(* Logix 5000 project; controller cal1632 1756-L62 rev 16.20; software revision 16.05; part 30 of 61 *)
(* tags used below, declared in another part *)
   AFI : BOOL;
   FAULT : BOOL;
   p01r02_plc_scan_time_in_sec : REAL;
   p01r09 : routine;
   p01r09_pb_global_reset : BOOL;
   p01r12_master_ramped_speed : REAL;
   p01r13_line_running : BOOL;
   p01r13_line_slow_ramp : BOOL;
   p01r13_permissive_drives : BOOL;
   p20_ai_lc01 : REAL;
   p20_ai_letoff_dia : REAL;
   p20_ai_lob_speed : REAL;
   p20_ao_lo_turret_selected_speed : REAL;
   p20_ao_lob_selected_speed : REAL;
   p20_ao_lob_torque : REAL;
   p20_di_clutch_prs_ok : BOOL;
   p20_di_lo_turret : acs800_di_normal;
   p20_di_lo_turret_therm : BOOL;
   p20_di_loa_active : BOOL;
   p20_di_lob_brake_thermostat : BOOL;
   p20_di_lob_fwd_dir : BOOL;
   p20_di_lob_jog : BOOL;
   p20_di_lob_motor_thermostat : BOOL;
   p20_di_lob_start : BOOL;
   p20_di_lob_stop : BOOL;
   p20_di_turret_fwd : BOOL;
   p20_di_turret_pos : BOOL;
   p20_di_turret_rev : BOOL;
   p20_do_close_nip : BOOL;
   p20_do_wdr_turret : acs800_do_normal;
   p20_param_high_accel_rate : REAL;
   p20_param_high_decel_rate : REAL;
   p20_param_jog_accel_rate : REAL;
   p20_param_jog_decel_rate : REAL;
   p20_param_letoff_jog_speed : REAL;
   p20_param_lo_turret_index_speed : REAL;
   p20_param_lof_fast_fill : REAL;
   p20_param_lof_slow_fill : REAL;
   p20_param_lof_stop_fill : REAL;
   p20_param_norm_accel_rate : REAL;
   p20_param_norm_decel_rate : REAL;
   p20_param_run_torque : REAL;
   p20_request_run_index_dir : BOOL;
   p20_request_run_index_rev_dir : BOOL;
   p20_vfd_di_lob : acs800_di_normal;
   p20_vfd_do_lob : acs800_do_normal;
   p20r10_speed_offset : REAL;
   p20r13_state : DINT;
   p20r15 : routine;
   p20r15_loa_on : BOOL;
   p20r15_request_tension : BOOL;
   p20r16 : routine;
   p20r16_loa_accel_decel_ramp : SYS_ACC_DEC_RAMP;
   p20r16_lob_accel : REAL;
   p20r16_lob_decel : REAL;
   p20r16_lob_on : BOOL;
   p20r16_lob_selected_speed : REAL;
   p20r16_permissive_run : BOOL;
   p20r16_request_jog_fwd : BOOL;
   p20r16_request_jog_rev : BOOL;
   p20r16_request_over_speed : BOOL;
   p20r16_request_position : BOOL;
   p20r16_request_stop : BOOL;
   p20r16_request_tension : BOOL;
   p20r16_request_thread_fwd : BOOL;
   p20r16_request_thread_rev : BOOL;
   p20r16_timer_fault : TIMER[10];
   p20r16_timer_warning : TIMER[4];
   p20r16_zero_speed : BOOL;
   p20r17 : routine;
   p20r17_ave_control : CONTROL;
   p20r17_diameter_clac_active : BOOL;
   p20r17_letoff_avg_diam_inch : REAL;
   p20r17_letoff_diam_avg_stack : REAL[20];
   p20r17_stack_ctrl : CONTROL;
   p20r17_timer : TIMER[5];
   p20r17_timer_fault : TIMER[5];
   p20r17_timer_warning : TIMER[5];
   p20r17_winder_a_unload : REAL;
   p20r18 : routine;
   p20r18_acc_dec_ramp : SYS_ACC_DEC_RAMP;
   p20r18_accel_rate : REAL;
   p20r18_decel_rate : REAL;
   p20r18_index_complete : BOOL;
   p20r18_index_move_timer : TIMER;
   p20r18_index_time : DINT;
   p20r18_index_time_offset : DINT;
   p20r18_index_timer : TIMER;
   p20r18_pb_index_fwd : BOOL;
   p20r18_pb_index_rev : BOOL;
   p20r18_permissive : BOOL;
   p20r18_request_index_fwd : BOOL;
   p20r18_request_index_rev : BOOL;
   p20r18_selected_speed : REAL;
   p20r18_timer_fault : TIMER[10];
   p20r18_timer_warning : TIMER[4];
   p20r18_zero_speed : BOOL;
   p22_ao_selected_speed : REAL;
   p22r11_request_thread_fwd : BOOL;
   p22r11_request_thread_rev : BOOL;
   p25r11_request_thread_fwd : BOOL;
   p25r11_request_thread_rev : BOOL;
(* P20_Letoff, continued *)

ROUTINE R16_Letoff_B_VFD   (* ladder *)
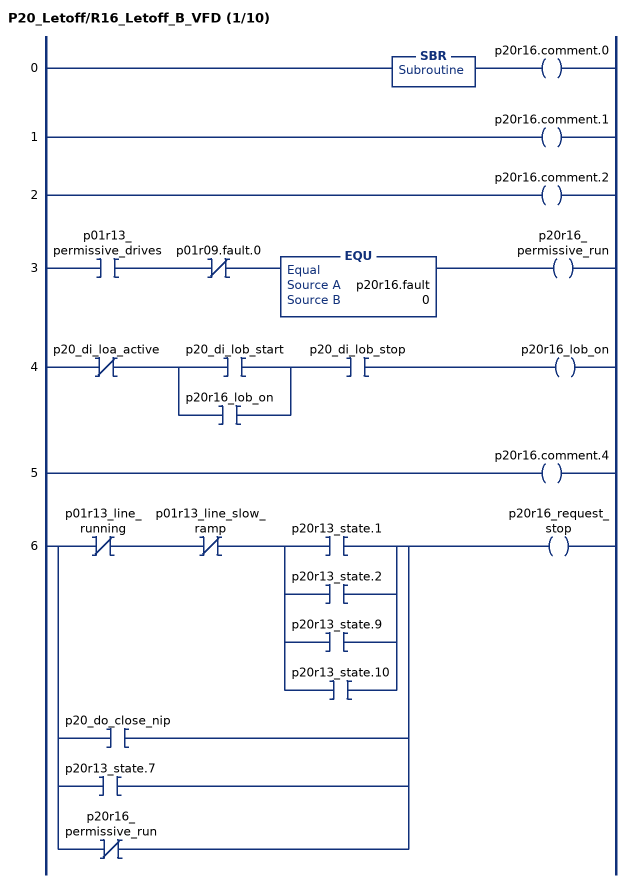
   0: SBR()OTE(p20r16.comment.0);
   1: OTE(p20r16.comment.1);
   2: OTE(p20r16.comment.2);
   3: XIC(p01r13_permissive_drives)XIO(p01r09.fault.0)EQU(p20r16.fault,0)OTE(p20r16_permissive_run);
   4: XIO(p20_di_loa_active)[XIC(p20_di_lob_start) ,XIC(p20r16_lob_on) ]XIC(p20_di_lob_stop)OTE(p20r16_lob_on);
   5: OTE(p20r16.comment.4);
   6: [XIO(p01r13_line_running) XIO(p01r13_line_slow_ramp) [XIC(p20r13_state.1) ,XIC(p20r13_state.2) ,XIC(p20r13_state.9) ,XIC(p20r13_state.10) ] ,XIC(p20_do_close_nip) ,XIC(p20r13_state.7) ,XIO(p20r16_permissive_run) ]OTE(p20r16_request_stop);
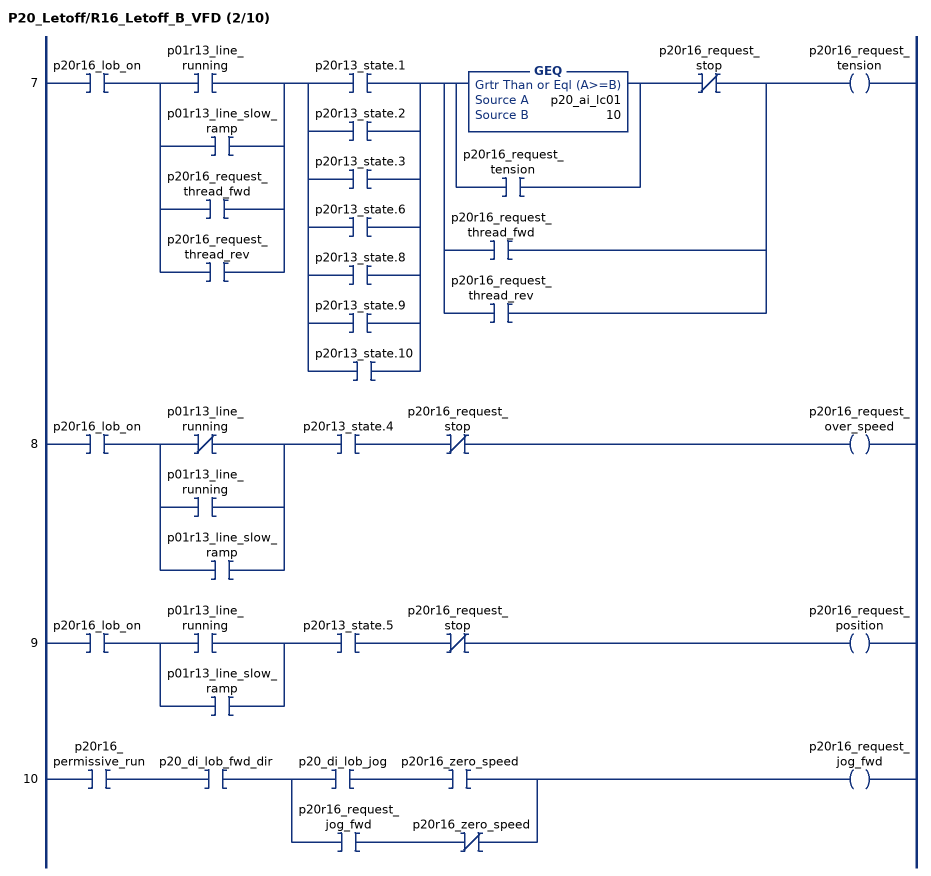
   7: XIC(p20r16_lob_on)[XIC(p01r13_line_running) ,XIC(p01r13_line_slow_ramp) ,XIC(p20r16_request_thread_fwd) ,XIC(p20r16_request_thread_rev) ][XIC(p20r13_state.1) ,XIC(p20r13_state.2) ,XIC(p20r13_state.3) ,XIC(p20r13_state.6) ,XIC(p20r13_state.8) ,XIC(p20r13_state.9) ,XIC(p20r13_state.10) ][[GEQ(p20_ai_lc01,10) ,XIC(p20r16_request_tension) ] XIO(p20r16_request_stop) ,XIC(p20r16_request_thread_fwd) ,XIC(p20r16_request_thread_rev) ]OTE(p20r16_request_tension);
   8: XIC(p20r16_lob_on)[XIO(p01r13_line_running) ,XIC(p01r13_line_running) ,XIC(p01r13_line_slow_ramp) ]XIC(p20r13_state.4)XIO(p20r16_request_stop)OTE(p20r16_request_over_speed);
   9: XIC(p20r16_lob_on)[XIC(p01r13_line_running) ,XIC(p01r13_line_slow_ramp) ]XIC(p20r13_state.5)XIO(p20r16_request_stop)OTE(p20r16_request_position);
   10: XIC(p20r16_permissive_run)XIC(p20_di_lob_fwd_dir)[XIC(p20_di_lob_jog) XIC(p20r16_zero_speed) ,XIC(p20r16_request_jog_fwd) XIO(p20r16_zero_speed) ]OTE(p20r16_request_jog_fwd);
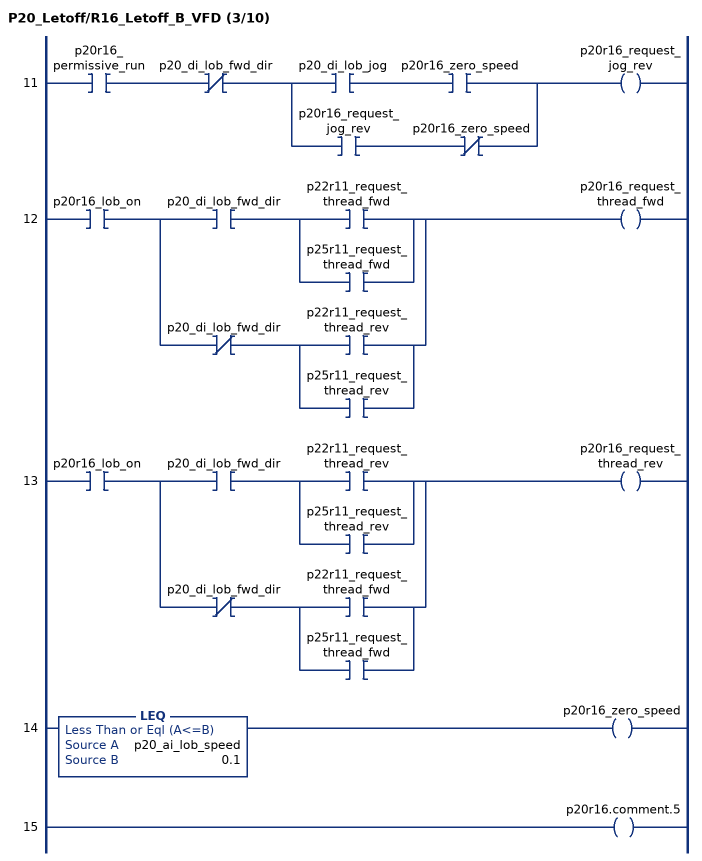
   11: XIC(p20r16_permissive_run)XIO(p20_di_lob_fwd_dir)[XIC(p20_di_lob_jog) XIC(p20r16_zero_speed) ,XIC(p20r16_request_jog_rev) XIO(p20r16_zero_speed) ]OTE(p20r16_request_jog_rev);
   12: XIC(p20r16_lob_on)[XIC(p20_di_lob_fwd_dir) [XIC(p22r11_request_thread_fwd) ,XIC(p25r11_request_thread_fwd) ] ,XIO(p20_di_lob_fwd_dir) [XIC(p22r11_request_thread_rev) ,XIC(p25r11_request_thread_rev) ] ]OTE(p20r16_request_thread_fwd);
   13: XIC(p20r16_lob_on)[XIC(p20_di_lob_fwd_dir) [XIC(p22r11_request_thread_rev) ,XIC(p25r11_request_thread_rev) ] ,XIO(p20_di_lob_fwd_dir) [XIC(p22r11_request_thread_fwd) ,XIC(p25r11_request_thread_fwd) ] ]OTE(p20r16_request_thread_rev);
   14: LEQ(p20_ai_lob_speed,0.1)OTE(p20r16_zero_speed);
   15: OTE(p20r16.comment.5);
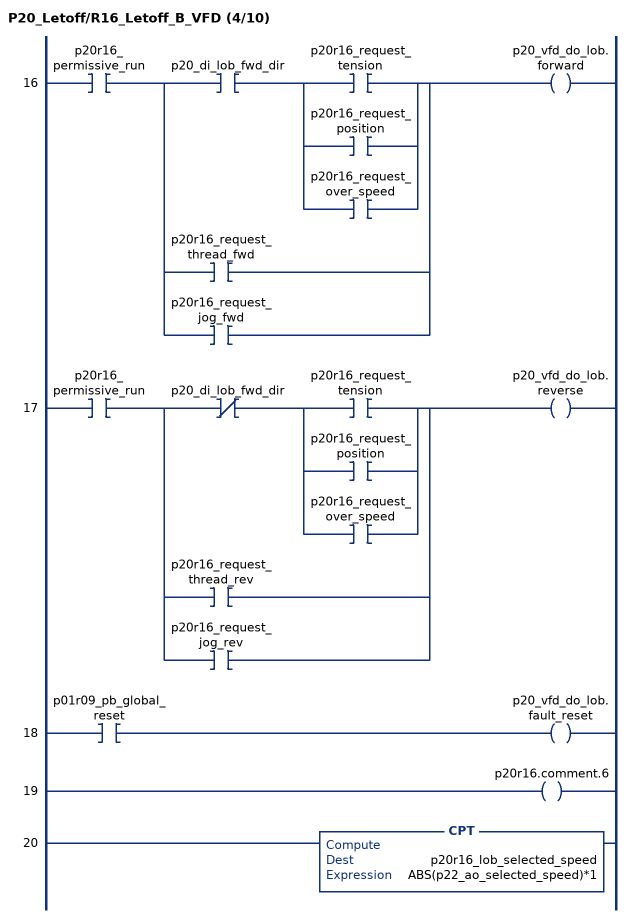
   16: XIC(p20r16_permissive_run)[XIC(p20_di_lob_fwd_dir) [XIC(p20r16_request_tension) ,XIC(p20r16_request_position) ,XIC(p20r16_request_over_speed) ] ,XIC(p20r16_request_thread_fwd) ,XIC(p20r16_request_jog_fwd) ]OTE(p20_vfd_do_lob.forward);
   17: XIC(p20r16_permissive_run)[XIO(p20_di_lob_fwd_dir) [XIC(p20r16_request_tension) ,XIC(p20r16_request_position) ,XIC(p20r16_request_over_speed) ] ,XIC(p20r16_request_thread_rev) ,XIC(p20r16_request_jog_rev) ]OTE(p20_vfd_do_lob.reverse);
   18: XIC(p01r09_pb_global_reset)OTE(p20_vfd_do_lob.fault_reset);
   19: OTE(p20r16.comment.6);
   20: CPT(p20r16_lob_selected_speed,ABS(p22_ao_selected_speed)*1);
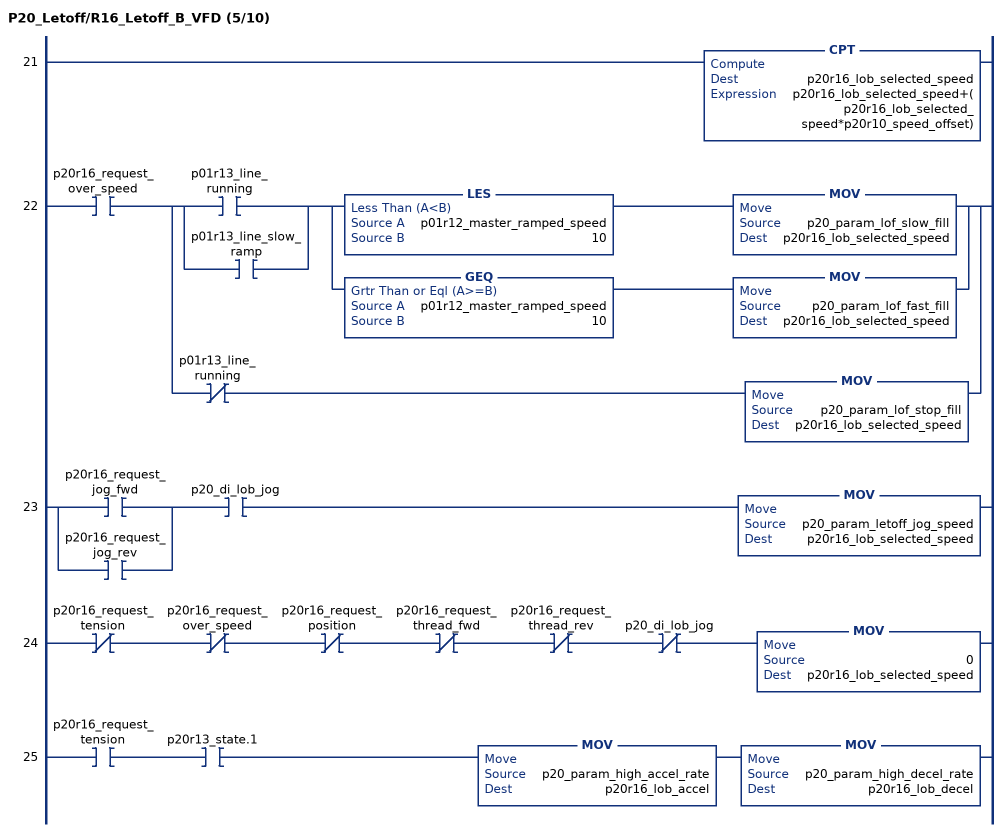
   21: CPT(p20r16_lob_selected_speed,p20r16_lob_selected_speed+(p20r16_lob_selected_speed*p20r10_speed_offset));
   22: XIC(p20r16_request_over_speed)[[XIC(p01r13_line_running) ,XIC(p01r13_line_slow_ramp) ] [LES(p01r12_master_ramped_speed,10) MOV(p20_param_lof_slow_fill,p20r16_lob_selected_speed) ,GEQ(p01r12_master_ramped_speed,10) MOV(p20_param_lof_fast_fill,p20r16_lob_selected_speed) ] ,XIO(p01r13_line_running) MOV(p20_param_lof_stop_fill,p20r16_lob_selected_speed) ];
   23: [XIC(p20r16_request_jog_fwd) ,XIC(p20r16_request_jog_rev) ]XIC(p20_di_lob_jog)MOV(p20_param_letoff_jog_speed,p20r16_lob_selected_speed);
   24: XIO(p20r16_request_tension)XIO(p20r16_request_over_speed)XIO(p20r16_request_position)XIO(p20r16_request_thread_fwd)XIO(p20r16_request_thread_rev)XIO(p20_di_lob_jog)MOV(0,p20r16_lob_selected_speed);
   25: XIC(p20r16_request_tension)XIC(p20r13_state.1)MOV(p20_param_high_accel_rate,p20r16_lob_accel)MOV(p20_param_high_decel_rate,p20r16_lob_decel);
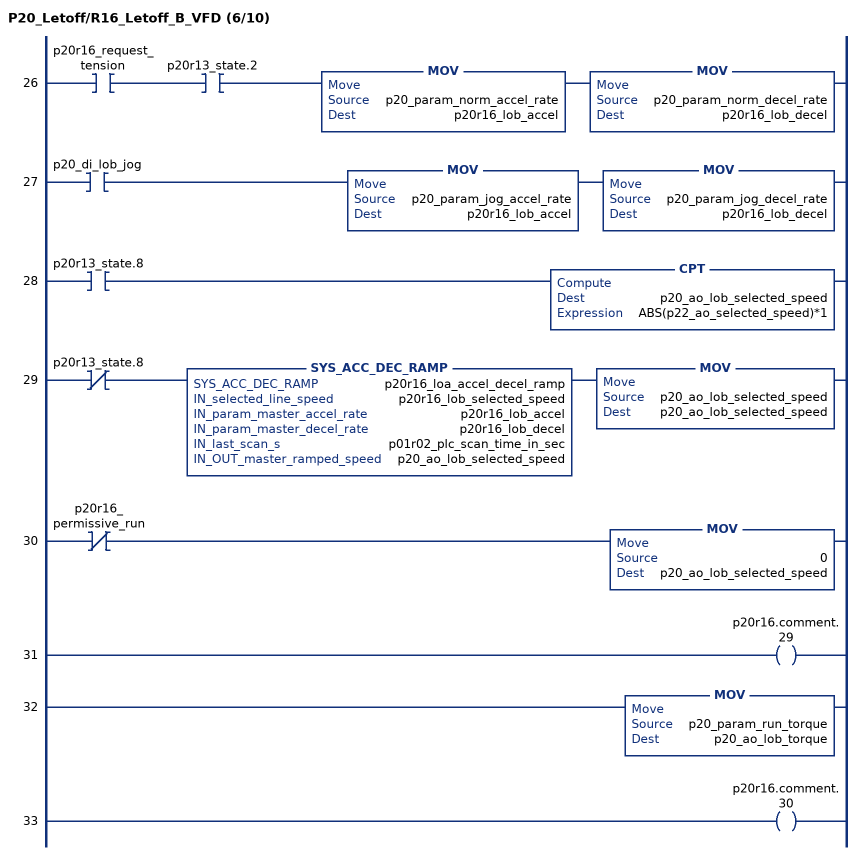
   26: XIC(p20r16_request_tension)XIC(p20r13_state.2)MOV(p20_param_norm_accel_rate,p20r16_lob_accel)MOV(p20_param_norm_decel_rate,p20r16_lob_decel);
   27: XIC(p20_di_lob_jog)MOV(p20_param_jog_accel_rate,p20r16_lob_accel)MOV(p20_param_jog_decel_rate,p20r16_lob_decel);
   28: XIC(p20r13_state.8)CPT(p20_ao_lob_selected_speed,ABS(p22_ao_selected_speed)*1);
   29: XIO(p20r13_state.8)SYS_ACC_DEC_RAMP(p20r16_loa_accel_decel_ramp,p20r16_lob_selected_speed,p20r16_lob_accel,p20r16_lob_decel,p01r02_plc_scan_time_in_sec,p20_ao_lob_selected_speed)MOV(p20_ao_lob_selected_speed,p20_ao_lob_selected_speed);
   30: XIO(p20r16_permissive_run)MOV(0,p20_ao_lob_selected_speed);
   31: OTE(p20r16.comment.29);
   32: MOV(p20_param_run_torque,p20_ao_lob_torque);
   33: OTE(p20r16.comment.30);
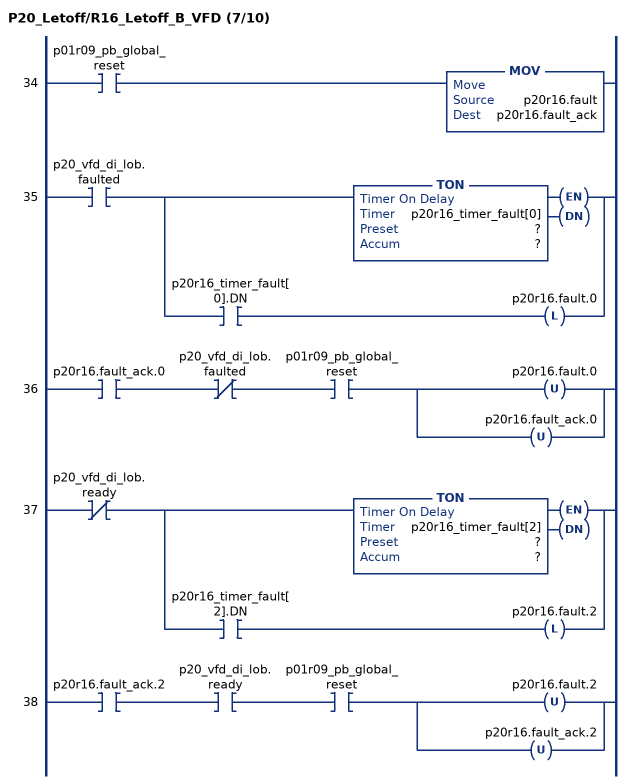
   34: XIC(p01r09_pb_global_reset)MOV(p20r16.fault,p20r16.fault_ack);
   35: XIC(p20_vfd_di_lob.faulted)[TON(p20r16_timer_fault[0],?,?) ,XIC(p20r16_timer_fault[0].DN) OTL(p20r16.fault.0) ];
   36: XIC(p20r16.fault_ack.0)XIO(p20_vfd_di_lob.faulted)XIC(p01r09_pb_global_reset)[OTU(p20r16.fault.0) ,OTU(p20r16.fault_ack.0) ];
   37: XIO(p20_vfd_di_lob.ready)[TON(p20r16_timer_fault[2],?,?) ,XIC(p20r16_timer_fault[2].DN) OTL(p20r16.fault.2) ];
   38: XIC(p20r16.fault_ack.2)XIC(p20_vfd_di_lob.ready)XIC(p01r09_pb_global_reset)[OTU(p20r16.fault.2) ,OTU(p20r16.fault_ack.2) ];
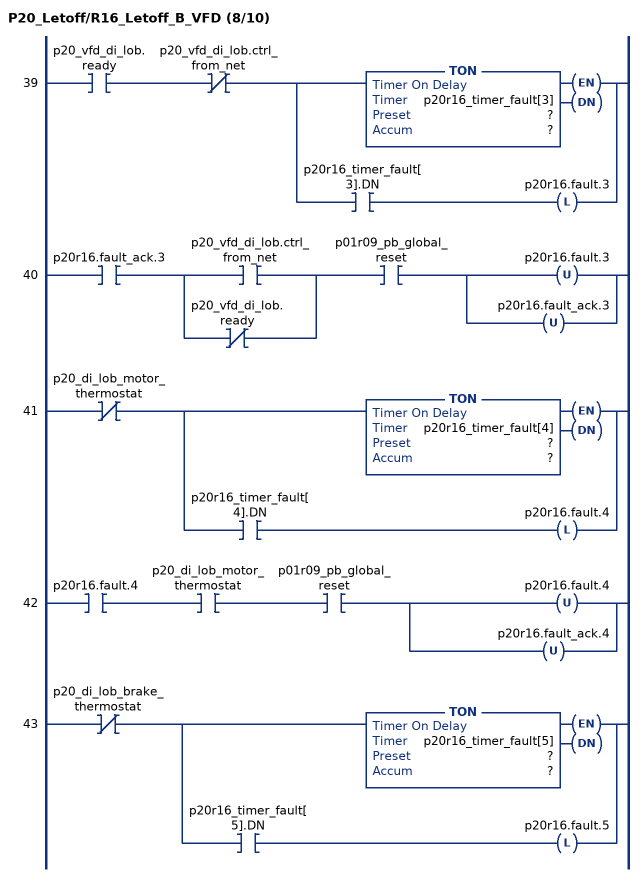
   39: XIC(p20_vfd_di_lob.ready)XIO(p20_vfd_di_lob.ctrl_from_net)[TON(p20r16_timer_fault[3],?,?) ,XIC(p20r16_timer_fault[3].DN) OTL(p20r16.fault.3) ];
   40: XIC(p20r16.fault_ack.3)[XIC(p20_vfd_di_lob.ctrl_from_net) ,XIO(p20_vfd_di_lob.ready) ]XIC(p01r09_pb_global_reset)[OTU(p20r16.fault.3) ,OTU(p20r16.fault_ack.3) ];
   41: XIO(p20_di_lob_motor_thermostat)[TON(p20r16_timer_fault[4],?,?) ,XIC(p20r16_timer_fault[4].DN) OTL(p20r16.fault.4) ];
   42: XIC(p20r16.fault.4)XIC(p20_di_lob_motor_thermostat)XIC(p01r09_pb_global_reset)[OTU(p20r16.fault.4) ,OTU(p20r16.fault_ack.4) ];
   43: XIO(p20_di_lob_brake_thermostat)[TON(p20r16_timer_fault[5],?,?) ,XIC(p20r16_timer_fault[5].DN) OTL(p20r16.fault.5) ];
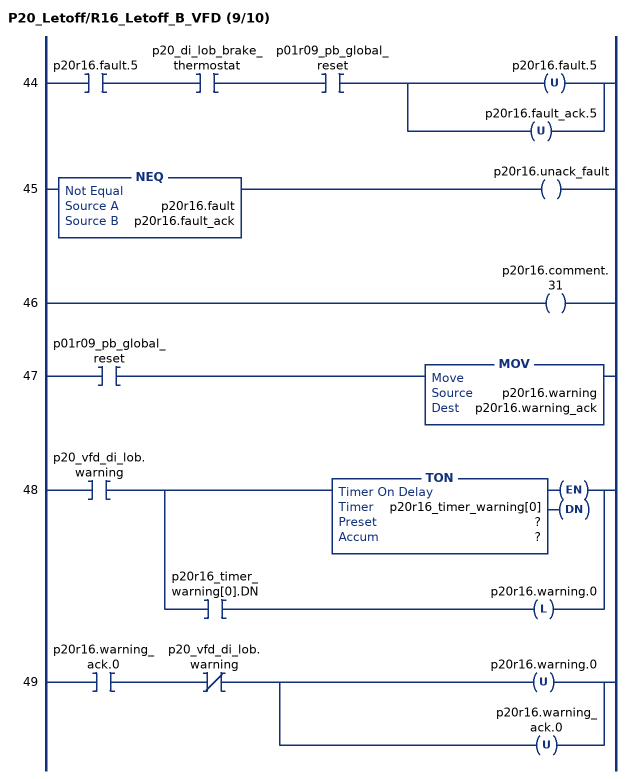
   44: XIC(p20r16.fault.5)XIC(p20_di_lob_brake_thermostat)XIC(p01r09_pb_global_reset)[OTU(p20r16.fault.5) ,OTU(p20r16.fault_ack.5) ];
   45: NEQ(p20r16.fault,p20r16.fault_ack)OTE(p20r16.unack_fault);
   46: OTE(p20r16.comment.31);
   47: XIC(p01r09_pb_global_reset)MOV(p20r16.warning,p20r16.warning_ack);
   48: XIC(p20_vfd_di_lob.warning)[TON(p20r16_timer_warning[0],?,?) ,XIC(p20r16_timer_warning[0].DN) OTL(p20r16.warning.0) ];
   49: XIC(p20r16.warning_ack.0)XIO(p20_vfd_di_lob.warning)[OTU(p20r16.warning.0) ,OTU(p20r16.warning_ack.0) ];
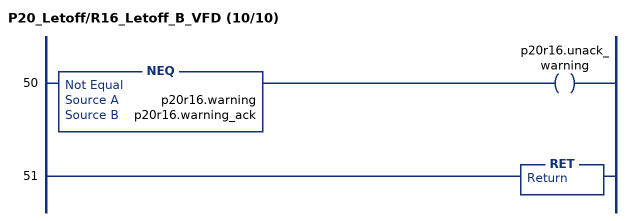
   50: NEQ(p20r16.warning,p20r16.warning_ack)OTE(p20r16.unack_warning);
   51: RET();
END_ROUTINE

ROUTINE R17_Letoff_Diameter_Calc   (* ladder *)
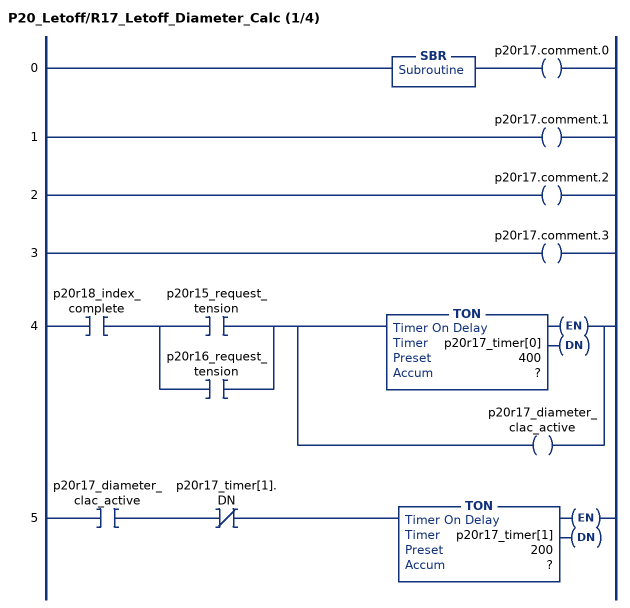
   0: SBR()OTE(p20r17.comment.0);
   1: OTE(p20r17.comment.1);
   2: OTE(p20r17.comment.2);
   3: OTE(p20r17.comment.3);
   4: XIC(p20r18_index_complete)[XIC(p20r15_request_tension) ,XIC(p20r16_request_tension) ][TON(p20r17_timer[0],?,?) ,OTE(p20r17_diameter_clac_active) ];
   5: XIC(p20r17_diameter_clac_active)XIO(p20r17_timer[1].DN)TON(p20r17_timer[1],?,?);
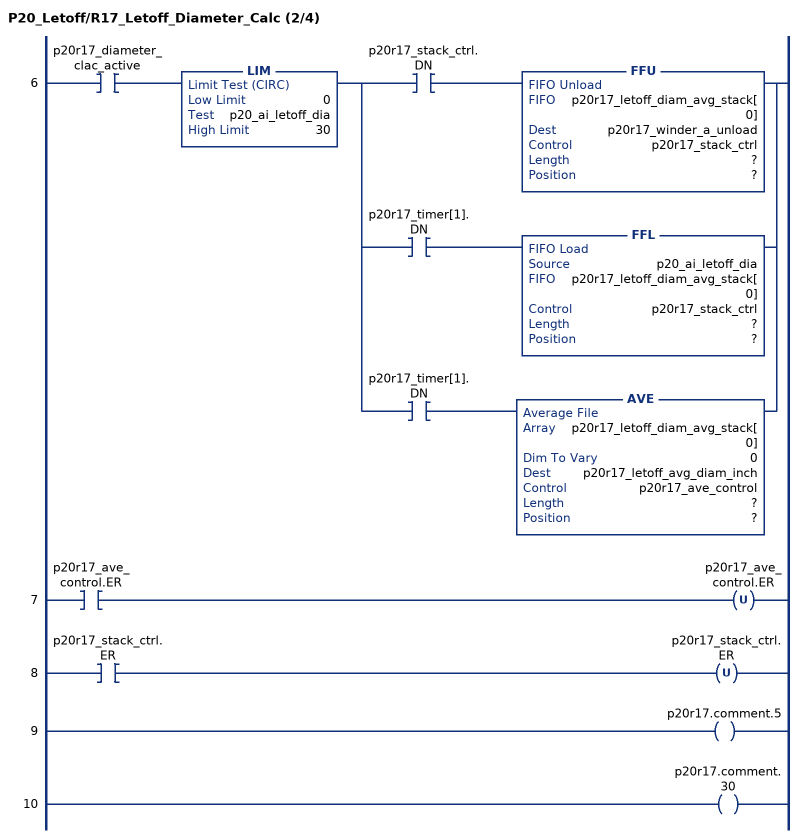
   6: XIC(p20r17_diameter_clac_active)LIM(0,p20_ai_letoff_dia,30)[XIC(p20r17_stack_ctrl.DN) FFU(p20r17_letoff_diam_avg_stack[0],p20r17_winder_a_unload,p20r17_stack_ctrl,?,?) ,XIC(p20r17_timer[1].DN) FFL(p20_ai_letoff_dia,p20r17_letoff_diam_avg_stack[0],p20r17_stack_ctrl,?,?) ,XIC(p20r17_timer[1].DN) AVE(p20r17_letoff_diam_avg_stack[0],0,p20r17_letoff_avg_diam_inch,p20r17_ave_control,?,?) ];
   7: XIC(p20r17_ave_control.ER)OTU(p20r17_ave_control.ER);
   8: XIC(p20r17_stack_ctrl.ER)OTU(p20r17_stack_ctrl.ER);
   9: OTE(p20r17.comment.5);
   10: OTE(p20r17.comment.30);
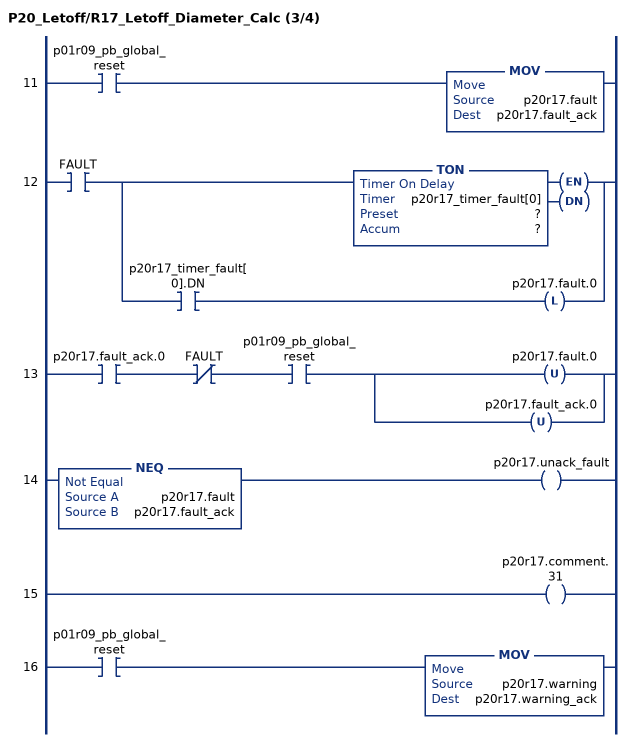
   11: XIC(p01r09_pb_global_reset)MOV(p20r17.fault,p20r17.fault_ack);
   12: XIC(FAULT)[TON(p20r17_timer_fault[0],?,?) ,XIC(p20r17_timer_fault[0].DN) OTL(p20r17.fault.0) ];
   13: XIC(p20r17.fault_ack.0)XIO(FAULT)XIC(p01r09_pb_global_reset)[OTU(p20r17.fault.0) ,OTU(p20r17.fault_ack.0) ];
   14: NEQ(p20r17.fault,p20r17.fault_ack)OTE(p20r17.unack_fault);
   15: OTE(p20r17.comment.31);
   16: XIC(p01r09_pb_global_reset)MOV(p20r17.warning,p20r17.warning_ack);
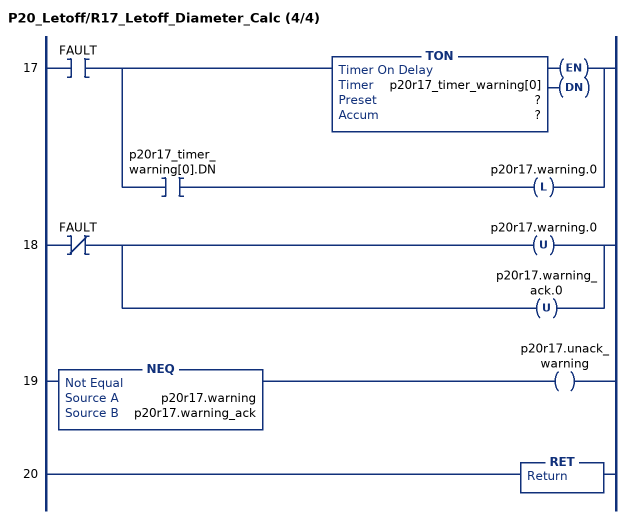
   17: XIC(FAULT)[TON(p20r17_timer_warning[0],?,?) ,XIC(p20r17_timer_warning[0].DN) OTL(p20r17.warning.0) ];
   18: XIO(FAULT)[OTU(p20r17.warning.0) ,OTU(p20r17.warning_ack.0) ];
   19: NEQ(p20r17.warning,p20r17.warning_ack)OTE(p20r17.unack_warning);
   20: RET();
END_ROUTINE

ROUTINE R18_Letoff_Turret_VFD   (* ladder *)
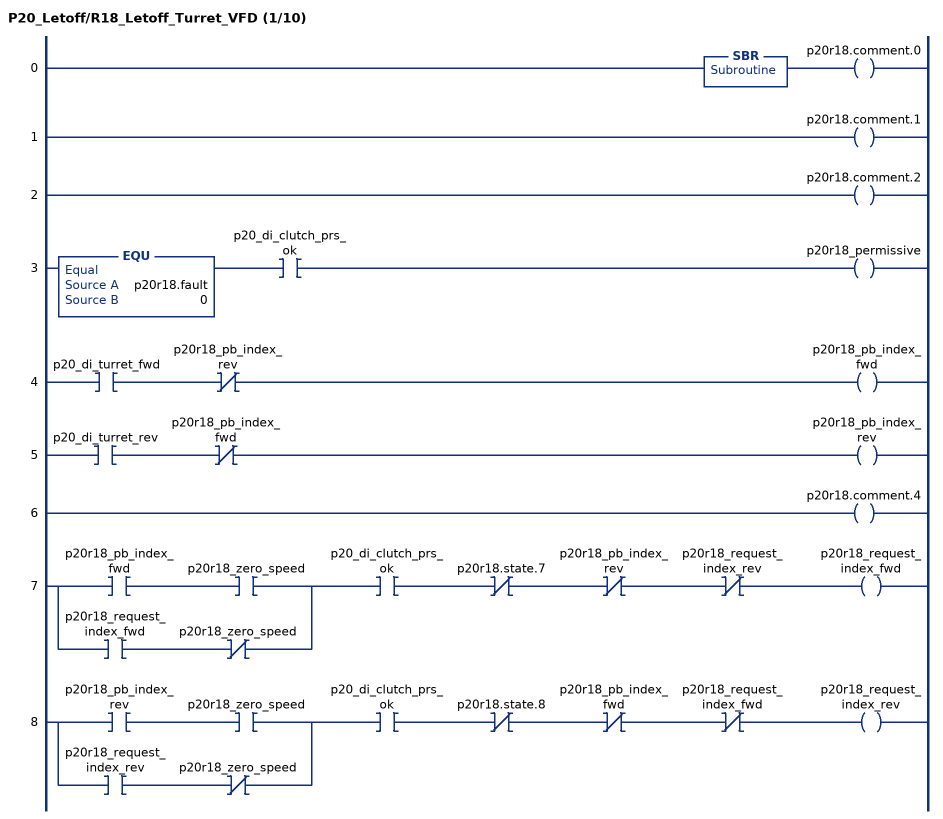
   0: SBR()OTE(p20r18.comment.0);
   1: OTE(p20r18.comment.1);
   2: OTE(p20r18.comment.2);
   3: EQU(p20r18.fault,0)XIC(p20_di_clutch_prs_ok)OTE(p20r18_permissive);
   4: XIC(p20_di_turret_fwd)XIO(p20r18_pb_index_rev)OTE(p20r18_pb_index_fwd);
   5: XIC(p20_di_turret_rev)XIO(p20r18_pb_index_fwd)OTE(p20r18_pb_index_rev);
   6: OTE(p20r18.comment.4);
   7: [XIC(p20r18_pb_index_fwd) XIC(p20r18_zero_speed) ,XIC(p20r18_request_index_fwd) XIO(p20r18_zero_speed) ]XIC(p20_di_clutch_prs_ok)XIO(p20r18.state.7)XIO(p20r18_pb_index_rev)XIO(p20r18_request_index_rev)OTE(p20r18_request_index_fwd);
   8: [XIC(p20r18_pb_index_rev) XIC(p20r18_zero_speed) ,XIC(p20r18_request_index_rev) XIO(p20r18_zero_speed) ]XIC(p20_di_clutch_prs_ok)XIO(p20r18.state.8)XIO(p20r18_pb_index_fwd)XIO(p20r18_request_index_fwd)OTE(p20r18_request_index_rev);
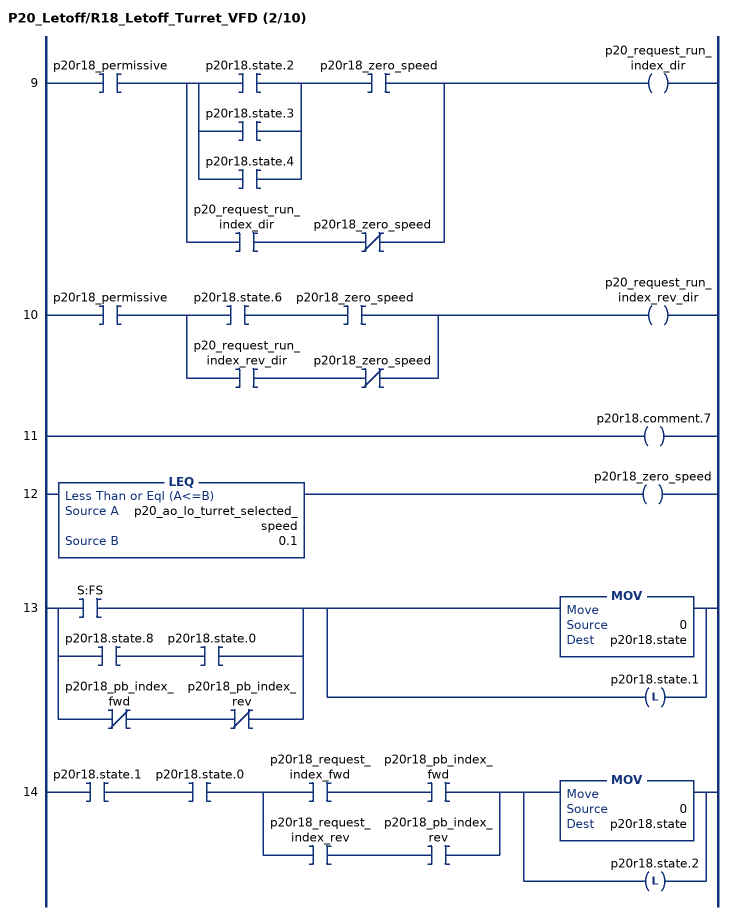
   9: XIC(p20r18_permissive)[[XIC(p20r18.state.2) ,XIC(p20r18.state.3) ,XIC(p20r18.state.4) ] XIC(p20r18_zero_speed) ,XIC(p20_request_run_index_dir) XIO(p20r18_zero_speed) ]OTE(p20_request_run_index_dir);
   10: XIC(p20r18_permissive)[XIC(p20r18.state.6) XIC(p20r18_zero_speed) ,XIC(p20_request_run_index_rev_dir) XIO(p20r18_zero_speed) ]OTE(p20_request_run_index_rev_dir);
   11: OTE(p20r18.comment.7);
   12: LEQ(p20_ao_lo_turret_selected_speed,0.1)OTE(p20r18_zero_speed);
   13: [XIC(S:FS) ,XIC(p20r18.state.8) XIC(p20r18.state.0) ,XIO(p20r18_pb_index_fwd) XIO(p20r18_pb_index_rev) ][MOV(0,p20r18.state) ,OTL(p20r18.state.1) ];
   14: XIC(p20r18.state.1)XIC(p20r18.state.0)[XIC(p20r18_request_index_fwd) XIC(p20r18_pb_index_fwd) ,XIC(p20r18_request_index_rev) XIC(p20r18_pb_index_rev) ][MOV(0,p20r18.state) ,OTL(p20r18.state.2) ];
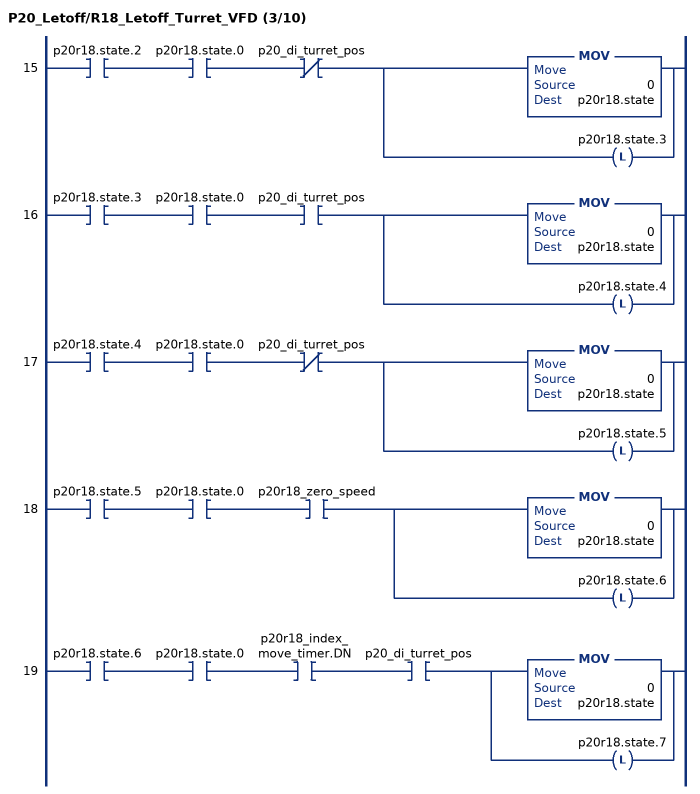
   15: XIC(p20r18.state.2)XIC(p20r18.state.0)XIO(p20_di_turret_pos)[MOV(0,p20r18.state) ,OTL(p20r18.state.3) ];
   16: XIC(p20r18.state.3)XIC(p20r18.state.0)XIC(p20_di_turret_pos)[MOV(0,p20r18.state) ,OTL(p20r18.state.4) ];
   17: XIC(p20r18.state.4)XIC(p20r18.state.0)XIO(p20_di_turret_pos)[MOV(0,p20r18.state) ,OTL(p20r18.state.5) ];
   18: XIC(p20r18.state.5)XIC(p20r18.state.0)XIC(p20r18_zero_speed)[MOV(0,p20r18.state) ,OTL(p20r18.state.6) ];
   19: XIC(p20r18.state.6)XIC(p20r18.state.0)XIC(p20r18_index_move_timer.DN)XIC(p20_di_turret_pos)[MOV(0,p20r18.state) ,OTL(p20r18.state.7) ];
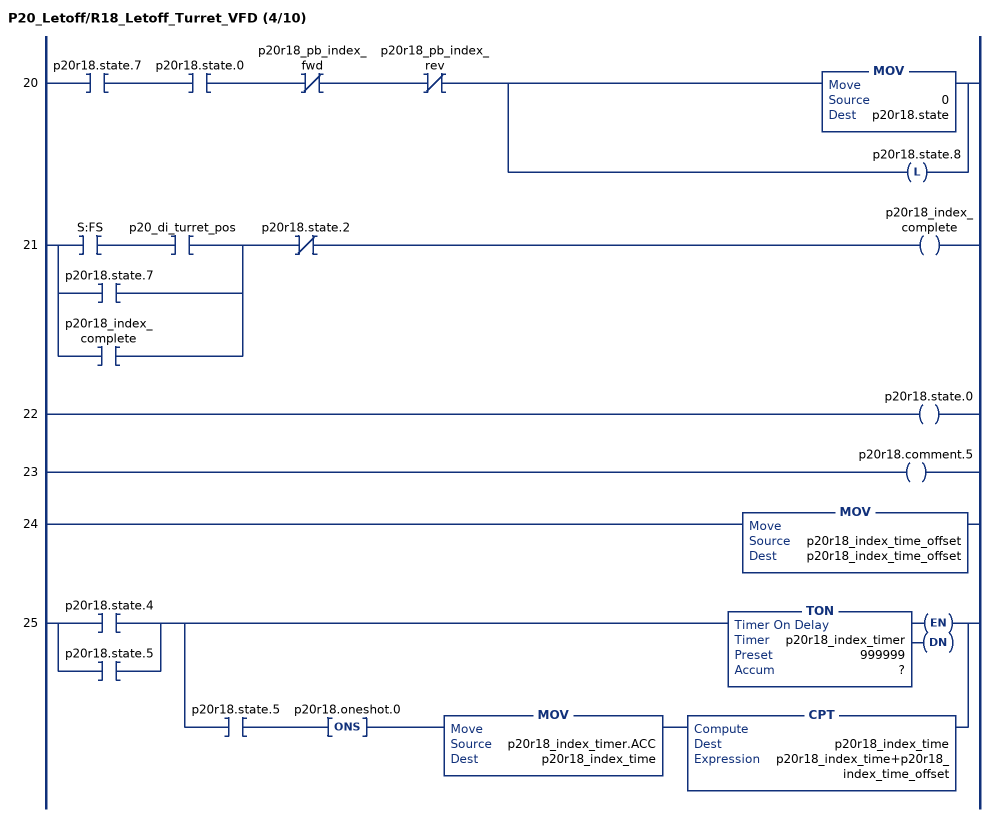
   20: XIC(p20r18.state.7)XIC(p20r18.state.0)XIO(p20r18_pb_index_fwd)XIO(p20r18_pb_index_rev)[MOV(0,p20r18.state) ,OTL(p20r18.state.8) ];
   21: [XIC(S:FS) XIC(p20_di_turret_pos) ,XIC(p20r18.state.7) ,XIC(p20r18_index_complete) ]XIO(p20r18.state.2)OTE(p20r18_index_complete);
   22: OTE(p20r18.state.0);
   23: OTE(p20r18.comment.5);
   24: MOV(p20r18_index_time_offset,p20r18_index_time_offset);
   25: [XIC(p20r18.state.4) ,XIC(p20r18.state.5) ][TON(p20r18_index_timer,?,?) ,XIC(p20r18.state.5) ONS(p20r18.oneshot.0) MOV(p20r18_index_timer.ACC,p20r18_index_time) CPT(p20r18_index_time,p20r18_index_time+p20r18_index_time_offset) ];
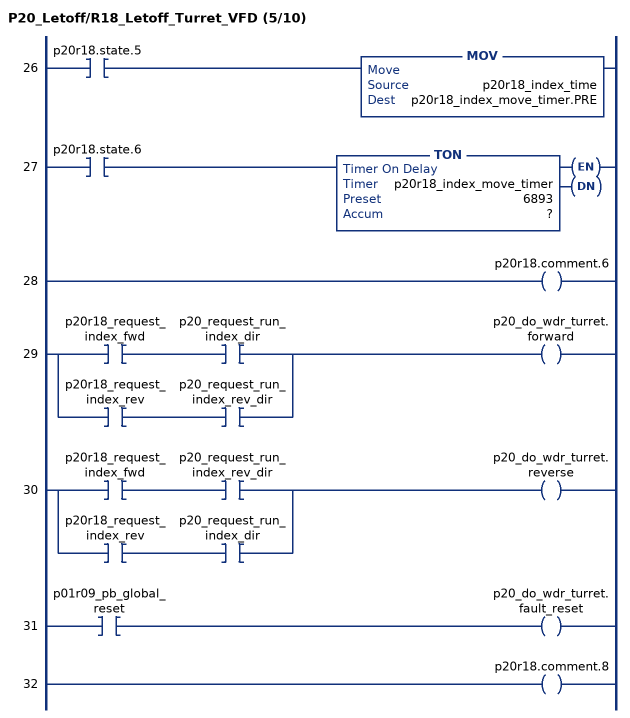
   26: XIC(p20r18.state.5)MOV(p20r18_index_time,p20r18_index_move_timer.PRE);
   27: XIC(p20r18.state.6)TON(p20r18_index_move_timer,?,?);
   28: OTE(p20r18.comment.6);
   29: [XIC(p20r18_request_index_fwd) XIC(p20_request_run_index_dir) ,XIC(p20r18_request_index_rev) XIC(p20_request_run_index_rev_dir) ]OTE(p20_do_wdr_turret.forward);
   30: [XIC(p20r18_request_index_fwd) XIC(p20_request_run_index_rev_dir) ,XIC(p20r18_request_index_rev) XIC(p20_request_run_index_dir) ]OTE(p20_do_wdr_turret.reverse);
   31: XIC(p01r09_pb_global_reset)OTE(p20_do_wdr_turret.fault_reset);
   32: OTE(p20r18.comment.8);
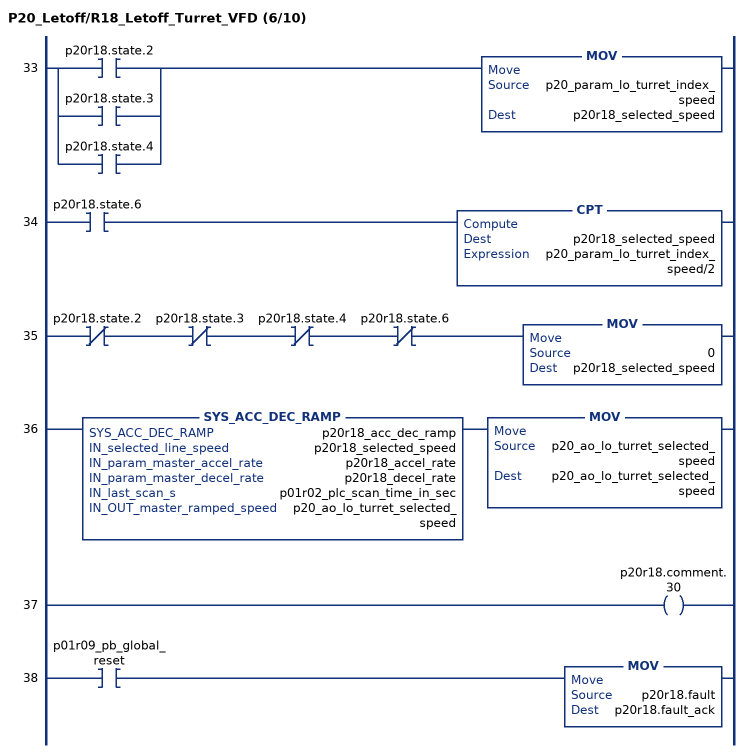
   33: [XIC(p20r18.state.2) ,XIC(p20r18.state.3) ,XIC(p20r18.state.4) ]MOV(p20_param_lo_turret_index_speed,p20r18_selected_speed);
   34: XIC(p20r18.state.6)CPT(p20r18_selected_speed,p20_param_lo_turret_index_speed/2);
   35: XIO(p20r18.state.2)XIO(p20r18.state.3)XIO(p20r18.state.4)XIO(p20r18.state.6)MOV(0,p20r18_selected_speed);
   36: SYS_ACC_DEC_RAMP(p20r18_acc_dec_ramp,p20r18_selected_speed,p20r18_accel_rate,p20r18_decel_rate,p01r02_plc_scan_time_in_sec,p20_ao_lo_turret_selected_speed)MOV(p20_ao_lo_turret_selected_speed,p20_ao_lo_turret_selected_speed);
   37: OTE(p20r18.comment.30);
   38: XIC(p01r09_pb_global_reset)MOV(p20r18.fault,p20r18.fault_ack);
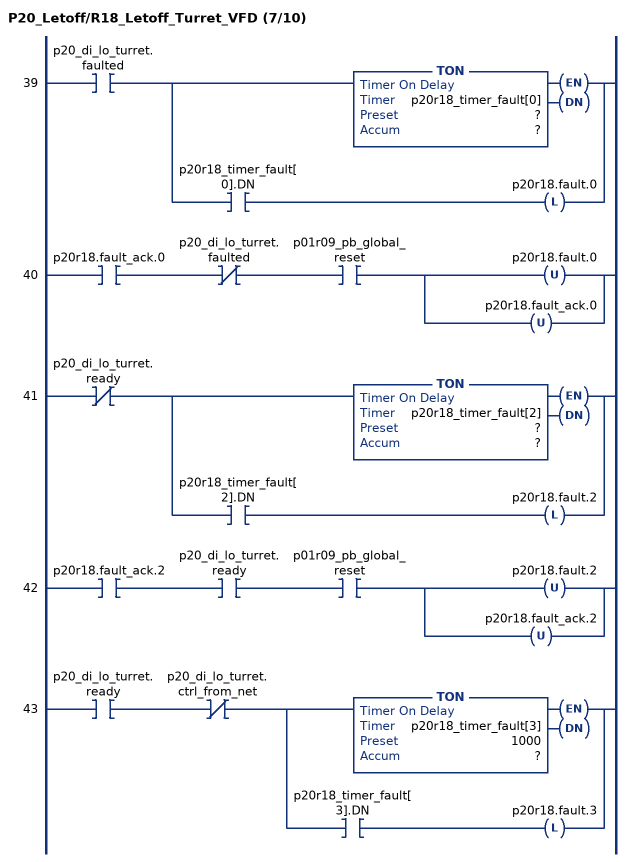
   39: XIC(p20_di_lo_turret.faulted)[TON(p20r18_timer_fault[0],?,?) ,XIC(p20r18_timer_fault[0].DN) OTL(p20r18.fault.0) ];
   40: XIC(p20r18.fault_ack.0)XIO(p20_di_lo_turret.faulted)XIC(p01r09_pb_global_reset)[OTU(p20r18.fault.0) ,OTU(p20r18.fault_ack.0) ];
   41: XIO(p20_di_lo_turret.ready)[TON(p20r18_timer_fault[2],?,?) ,XIC(p20r18_timer_fault[2].DN) OTL(p20r18.fault.2) ];
   42: XIC(p20r18.fault_ack.2)XIC(p20_di_lo_turret.ready)XIC(p01r09_pb_global_reset)[OTU(p20r18.fault.2) ,OTU(p20r18.fault_ack.2) ];
   43: XIC(p20_di_lo_turret.ready)XIO(p20_di_lo_turret.ctrl_from_net)[TON(p20r18_timer_fault[3],?,?) ,XIC(p20r18_timer_fault[3].DN) OTL(p20r18.fault.3) ];
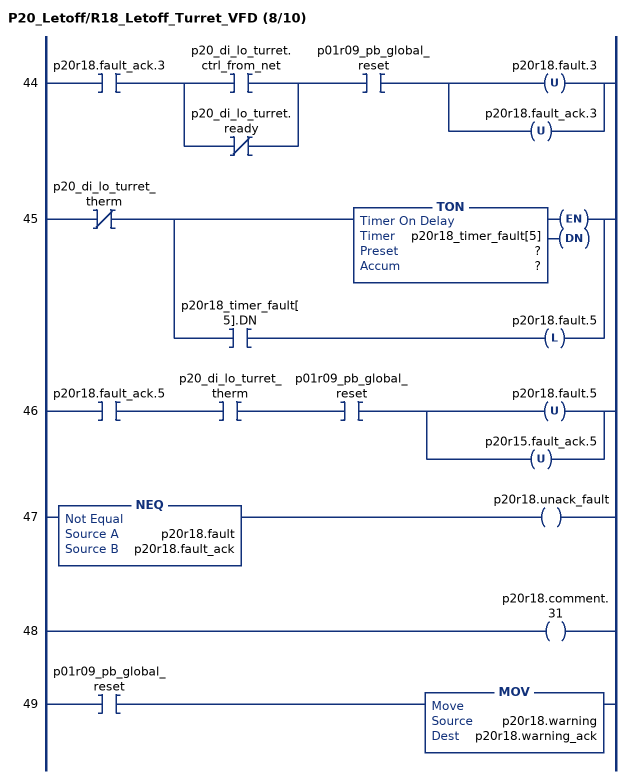
   44: XIC(p20r18.fault_ack.3)[XIC(p20_di_lo_turret.ctrl_from_net) ,XIO(p20_di_lo_turret.ready) ]XIC(p01r09_pb_global_reset)[OTU(p20r18.fault.3) ,OTU(p20r18.fault_ack.3) ];
   45: XIO(p20_di_lo_turret_therm)[TON(p20r18_timer_fault[5],?,?) ,XIC(p20r18_timer_fault[5].DN) OTL(p20r18.fault.5) ];
   46: XIC(p20r18.fault_ack.5)XIC(p20_di_lo_turret_therm)XIC(p01r09_pb_global_reset)[OTU(p20r18.fault.5) ,OTU(p20r15.fault_ack.5) ];
   47: NEQ(p20r18.fault,p20r18.fault_ack)OTE(p20r18.unack_fault);
   48: OTE(p20r18.comment.31);
   49: XIC(p01r09_pb_global_reset)MOV(p20r18.warning,p20r18.warning_ack);
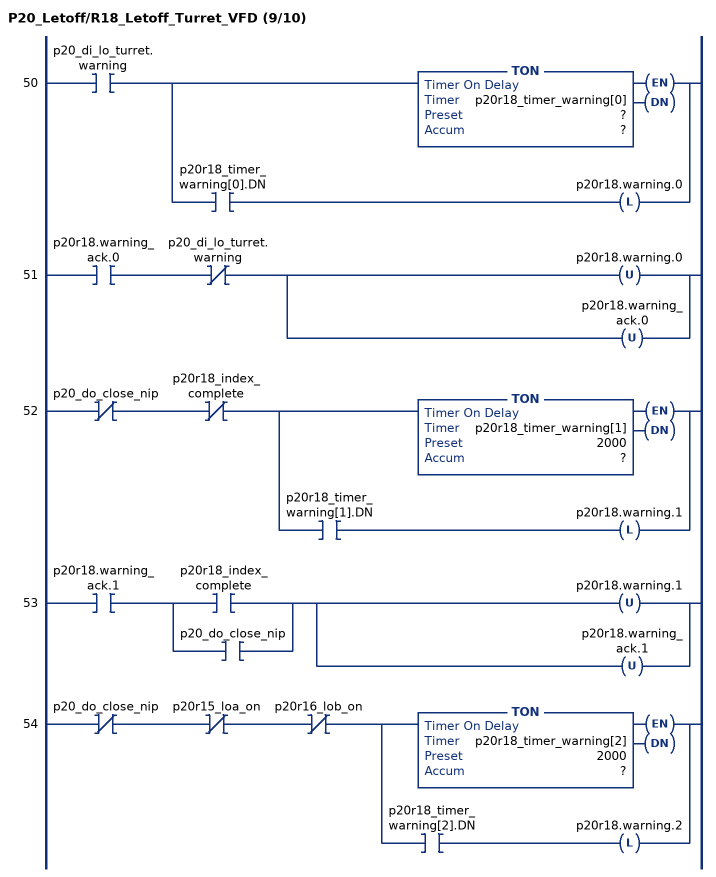
   50: XIC(p20_di_lo_turret.warning)[TON(p20r18_timer_warning[0],?,?) ,XIC(p20r18_timer_warning[0].DN) OTL(p20r18.warning.0) ];
   51: XIC(p20r18.warning_ack.0)XIO(p20_di_lo_turret.warning)[OTU(p20r18.warning.0) ,OTU(p20r18.warning_ack.0) ];
   52: XIO(p20_do_close_nip)XIO(p20r18_index_complete)[TON(p20r18_timer_warning[1],?,?) ,XIC(p20r18_timer_warning[1].DN) OTL(p20r18.warning.1) ];
   53: XIC(p20r18.warning_ack.1)[XIC(p20r18_index_complete) ,XIC(p20_do_close_nip) ][OTU(p20r18.warning.1) ,OTU(p20r18.warning_ack.1) ];
   54: XIO(p20_do_close_nip)XIO(p20r15_loa_on)XIO(p20r16_lob_on)[TON(p20r18_timer_warning[2],?,?) ,XIC(p20r18_timer_warning[2].DN) OTL(p20r18.warning.2) ];
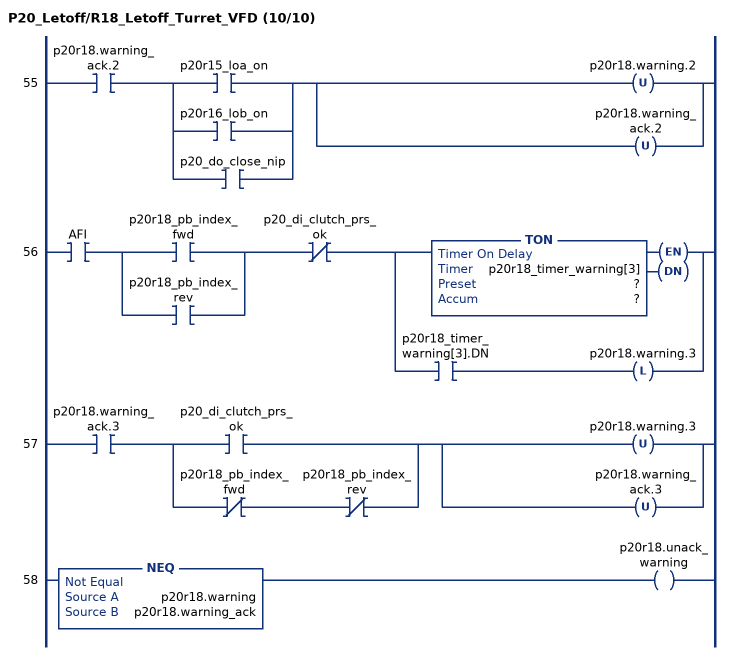
   55: XIC(p20r18.warning_ack.2)[XIC(p20r15_loa_on) ,XIC(p20r16_lob_on) ,XIC(p20_do_close_nip) ][OTU(p20r18.warning.2) ,OTU(p20r18.warning_ack.2) ];
   56: XIC(AFI)[XIC(p20r18_pb_index_fwd) ,XIC(p20r18_pb_index_rev) ]XIO(p20_di_clutch_prs_ok)[TON(p20r18_timer_warning[3],?,?) ,XIC(p20r18_timer_warning[3].DN) OTL(p20r18.warning.3) ];
   57: XIC(p20r18.warning_ack.3)[XIC(p20_di_clutch_prs_ok) ,XIO(p20r18_pb_index_fwd) XIO(p20r18_pb_index_rev) ][OTU(p20r18.warning.3) ,OTU(p20r18.warning_ack.3) ];
   58: NEQ(p20r18.warning,p20r18.warning_ack)OTE(p20r18.unack_warning);
END_ROUTINE
END_PROGRAM
